# EPICS autosave request: ThorLabsDFMApp/Db/ThorLabsDFM_settings.req
$(P)$(R)ReadStatus.SCAN
$(P)$(R)SetTiltAmplitude
$(P)$(R)SetTiltAngle
